//Fills an array of LREAL of varible length with zeros
FUNCTION ZEROS
VAR_IN_OUT
	arr: ARRAY [*] OF LREAL;
END_VAR

FILL(arr := arr,val := 0.0);

END_FUNCTION

(* stored: Version 1.1.0.1, ProductVersion 3.1.4024.11
   POU ZEROS: Id {449177e9-991c-40f0-879f-55ab898b2896}, SpecialFunc None *)
